FUNCTION_BLOCK FB_BasicStatsFuns
VAR_INPUT
END_VAR
VAR_OUTPUT
END_VAR
VAR
END_VAR

METHOD M_Avg : LREAL
VAR_IN_OUT
	a : ARRAY[*] OF LREAL;
END_VAR

VAR
	upper: DINT;
	lower: DINT;
	sum:LREAL;
	idx:DINT;
	qtt: LREAL;
	avg: LREAL;
END_VAR
upper:=UPPER_BOUND(a,1);
lower:=LOWER_BOUND(a,1);

qtt:= DINT_TO_LREAL(upper-lower+1);

sum:=0;
FOR idx:=lower TO upper DO
	sum:= sum + a[idx];
END_FOR
IF qtt <> 0 THEN
	avg:= sum/qtt;
END_IF
M_Avg:=avg;
END_METHOD

METHOD M_Max : LREAL
VAR_IN_OUT
	a:ARRAY[*] OF LREAL;
END_VAR
VAR
	maximum:LREAL;
	upper: DINT;
	lower: DINT;
	range: LREAL;
	idx: DINT;
END_VAR
upper:=UPPER_BOUND(a,1);
lower:=LOWER_BOUND(a,1);

range:= DINT_TO_LREAL(upper-lower+1);

maximum:= a[lower];

FOR idx:= lower TO upper DO
	maximum:= MAX(maximum, a[idx]);
END_FOR
M_Max:= maximum;
END_METHOD

METHOD M_Min : LREAL
VAR_IN_OUT
	a:ARRAY[*] OF LREAL;
END_VAR
VAR
	minimum:LREAL;
	upper: DINT;
	lower: DINT;
	range: LREAL;
	idx: DINT;	
END_VAR
upper:=UPPER_BOUND(a,1);
lower:=LOWER_BOUND(a,1);

range:= DINT_TO_LREAL(upper-lower+1);

minimum:= a[lower];

FOR idx:= lower TO upper DO
	minimum:= MIN(minimum, a[idx]);
END_FOR
M_Min:= minimum;
END_METHOD

METHOD M_Range : LREAL
VAR_IN_OUT
	a:ARRAY[*] OF LREAL;
END_VAR
VAR
	maximum, minimum, range:LREAL;
END_VAR
maximum:= M_Max(a);
minimum:= M_Min(a);

range:= maximum-minimum;
M_Range:= range;
END_METHOD

METHOD M_Std : LREAL
VAR_IN_OUT
	a : ARRAY[*] OF LREAL;
END_VAR
VAR
	variance:LREAL;
	std:LREAL;
END_VAR
variance:= M_Variance(a);
std:= SQRT(variance);
M_Std:=std;
END_METHOD

METHOD M_Variance : LREAL
VAR_IN_OUT
	a : ARRAY[*] OF LREAL;
END_VAR
VAR
	avg, qtt:lreal;
	upper: DINT;
	lower: DINT;
	idx: DINT;
	numerator:LREAL;
END_VAR
upper:=UPPER_BOUND(a,1);
lower:=LOWER_BOUND(a,1);

qtt:= DINT_TO_LREAL(upper-lower+1);

avg:=M_Avg(a);
numerator:=0;

FOR idx:= lower TO upper DO
	numerator:= numerator+ EXPT(a[idx]-avg,2);
END_FOR

IF qtt <> 0 THEN
	M_Variance:= numerator/qtt;
END_IF
END_METHOD

END_FUNCTION_BLOCK

(* stored: Version 1.1.0.1, ProductVersion 3.1.4026.12
   POU FB_BasicStatsFuns: Id {3fa0b973-eb3e-4a78-90f3-2dea6596f72b}, SpecialFunc None
   Method M_Avg: Id {f85c6aff-3924-4e01-bd06-569ad7d41f51}
   Method M_Max: Id {307b30ef-7b30-4b7d-bb3c-b632073576a4}
   Method M_Min: Id {6aca99c8-5ac7-4861-9271-9fc7de40a6b5}
   Method M_Range: Id {5e15762d-8504-4b72-a79d-db2d965d9bc6}
   Method M_Std: Id {1871388c-8835-494c-aebb-c9b18b785abf}
   Method M_Variance: Id {c42ba802-e19a-4b53-9b4b-20a0d220991a} *)
